// TIA Portal V16 export
// export: Created 2021-11-12T13:32:58.6971257Z, ExportSetting WithDefaults, DisplayName Totally Integrated Automation Portal, DisplayVersion V16 Update 3, DisplayName TIA Portal Version Control Interface, DisplayVersion V16 Update 2, DisplayName TIA Portal Openness, DisplayVersion V16 Update 3, DisplayName SINAMICS Startdrive Advanced, DisplayVersion V16 Update 5, DisplayName SINAMICS Startdrive G130, G150, S120, S150, SINAMICS MV, S210, DisplayVersion V16 Update 5, DisplayName SINAMICS Startdrive G110M, G120, G120C, G120D, G120P, G115D, DisplayVersion V16 Update 5, DisplayName STEP 7 Professional, DisplayVersion V16 Update 3, DisplayName STEP 7 Safety, DisplayVersion V16, DisplayName WinCC UA Professional, DisplayVersion V16 Update 3
FUNCTION_BLOCK "StationTHM1"   // FB80, LAD
{ S7_Optimized_Access := 'TRUE' }
VERSION : 0.1
// stored: AutoNumber true, IsIECCheckEnabled false, IsRetainMemResEnabled false, MemoryReserve 100, SetENOAutomatically false, UDAEnableTagReadback false
   VAR_INPUT
      IS_Inputs : "UDT_COMM_THM1_CRS";   // Input structure from blasting machine THM1
   END_VAR
   VAR_OUTPUT
      OS_Outputs : "UDT_COMM_CRS_THM1";   // Output structure for blasting machine THM1
      OS_Specific : "UDT_THM_Status_specific";   // Specific output structure for blasting machine THM1
   END_VAR
   VAR
      SF_Alarm1 : "STD_DI_Mon";
      SF_Alarm2 : "STD_DI_Mon";
      SF_Alarm3 : "STD_DI_Mon";
      SF_Alarm4 : "STD_DI_Mon";
      SF_Alarm5 : "STD_DI_Mon";
      SF_Alarm6 : "STD_DI_Mon";
      SF_Alarm7 : "STD_DI_Mon";
      SF_Alarm8 : "STD_DI_Mon";
      SS_Edge : Array[0..15] of Bool;   // Edge evalution
      SS_ParamTemp : Struct   // Structure of parameters
         PartType : Int;   // Conveyor speed setpoint
         ConvSpd : Int;   // THM1 - Transportation system speed setpoint
      END_STRUCT;
      SB1ParamChanged : Bool;   // Production paramaters changed trigger
   END_VAR
   VAR_TEMP
      TB1PwrOk : Bool;   // Station powered
      TB1SetParam : Bool;   // Set loaded parameters memory
   END_VAR
   VAR_TEMP   // added for the SCL form of the ladder/FBD networks
      _w1 : Bool;
      _w2 : Bool;
   END_VAR
BEGIN

REGION Network 1: *************** Alarms ***************
END_REGION

REGION Network 2: Power OK
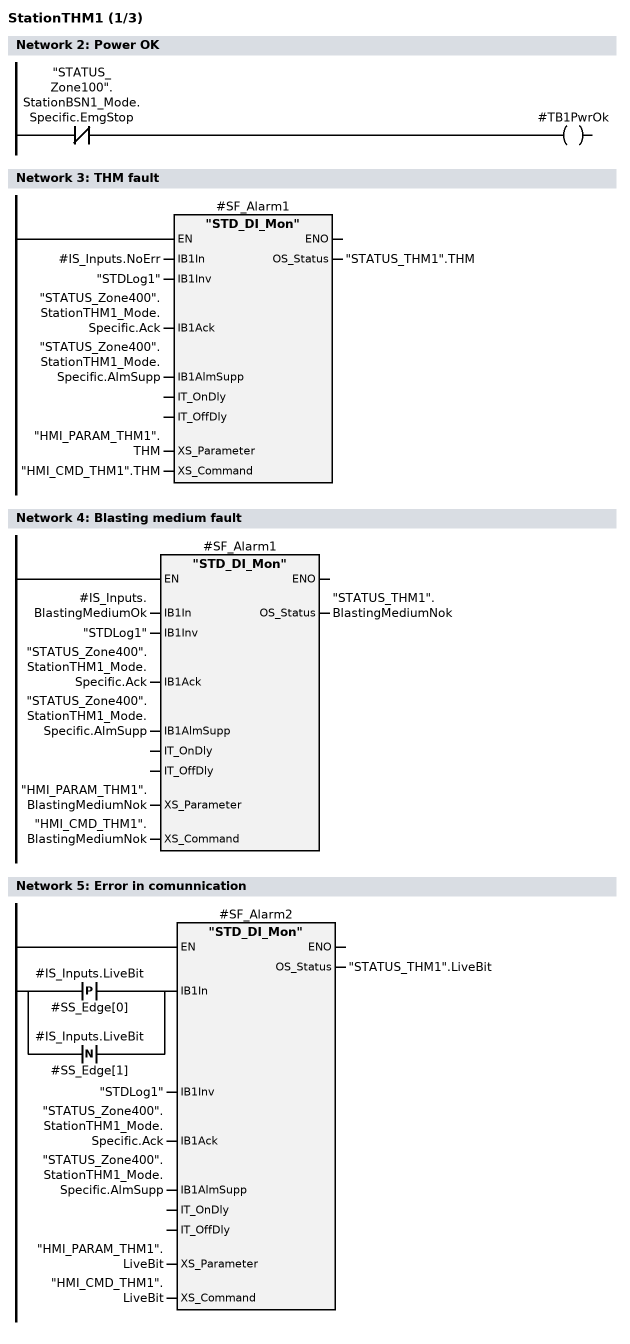
   RUNG wire#powerrail
      I_Contact( "STATUS_Zone100".StationBSN1_Mode.Specific.EmgStop )
      Coil( #TB1PwrOk )
   END_RUNG
   // the same network as SCL:
   #TB1PwrOk := NOT "STATUS_Zone100".StationBSN1_Mode.Specific.EmgStop;
END_REGION

REGION Network 3: THM fault
   RUNG wire#powerrail
      #SF_Alarm1(IB1In := #IS_Inputs.NoErr, IB1Inv := "STDLog1", IB1Ack := "STATUS_Zone400".StationTHM1_Mode.Specific.Ack, IB1AlmSupp := "STATUS_Zone400".StationTHM1_Mode.Specific.AlmSupp, IT_OnDly :=, IT_OffDly :=, XS_Parameter := "HMI_PARAM_THM1".THM, XS_Command := "HMI_CMD_THM1".THM, OS_Status => "STATUS_THM1".THM)
   END_RUNG
   // the same network as SCL:
   #SF_Alarm1(IB1In := #IS_Inputs.NoErr,   // "STD_DI_Mon"
              IB1Inv := "STDLog1",
              IB1Ack := "STATUS_Zone400".StationTHM1_Mode.Specific.Ack,
              IB1AlmSupp := "STATUS_Zone400".StationTHM1_Mode.Specific.AlmSupp,
              XS_Parameter := "HMI_PARAM_THM1".THM,
              XS_Command := "HMI_CMD_THM1".THM,
              OS_Status => "STATUS_THM1".THM);
END_REGION

REGION Network 4: Blasting medium fault
   RUNG wire#powerrail
      #SF_Alarm1(IB1In := #IS_Inputs.BlastingMediumOk, IB1Inv := "STDLog1", IB1Ack := "STATUS_Zone400".StationTHM1_Mode.Specific.Ack, IB1AlmSupp := "STATUS_Zone400".StationTHM1_Mode.Specific.AlmSupp, IT_OnDly :=, IT_OffDly :=, XS_Parameter := "HMI_PARAM_THM1".BlastingMediumNok, XS_Command := "HMI_CMD_THM1".BlastingMediumNok, OS_Status => "STATUS_THM1".BlastingMediumNok)
   END_RUNG
   // the same network as SCL:
   #SF_Alarm1(IB1In := #IS_Inputs.BlastingMediumOk,   // "STD_DI_Mon"
              IB1Inv := "STDLog1",
              IB1Ack := "STATUS_Zone400".StationTHM1_Mode.Specific.Ack,
              IB1AlmSupp := "STATUS_Zone400".StationTHM1_Mode.Specific.AlmSupp,
              XS_Parameter := "HMI_PARAM_THM1".BlastingMediumNok,
              XS_Command := "HMI_CMD_THM1".BlastingMediumNok,
              OS_Status => "STATUS_THM1".BlastingMediumNok);
END_REGION

REGION Network 5: Error in comunnication
   RUNG wire#powerrail
      #SF_Alarm2(IB1In := wire#w1, IB1Inv := "STDLog1", IB1Ack := "STATUS_Zone400".StationTHM1_Mode.Specific.Ack, IB1AlmSupp := "STATUS_Zone400".StationTHM1_Mode.Specific.AlmSupp, IT_OnDly :=, IT_OffDly :=, XS_Parameter := "HMI_PARAM_THM1".LiveBit, XS_Command := "HMI_CMD_THM1".LiveBit, OS_Status => "STATUS_THM1".LiveBit)
   END_RUNG
   RUNG wire#powerrail
      P_Contact(operand := #IS_Inputs.LiveBit, bit := #SS_Edge[0])
   END_RUNG wire#w1
   RUNG wire#powerrail
      N_Contact(operand := #IS_Inputs.LiveBit, bit := #SS_Edge[1])
   END_RUNG wire#w1
   // the same network as SCL:
   #_w1 := #IS_Inputs.LiveBit AND NOT #SS_Edge[0];   // rising edge of #IS_Inputs.LiveBit
   #SS_Edge[0] := #IS_Inputs.LiveBit;
   #_w2 := NOT #IS_Inputs.LiveBit AND #SS_Edge[1];   // falling edge of #IS_Inputs.LiveBit
   #SS_Edge[1] := #IS_Inputs.LiveBit;
   #SF_Alarm2(IB1In := #_w1 OR #_w2,   // "STD_DI_Mon"
              IB1Inv := "STDLog1",
              IB1Ack := "STATUS_Zone400".StationTHM1_Mode.Specific.Ack,
              IB1AlmSupp := "STATUS_Zone400".StationTHM1_Mode.Specific.AlmSupp,
              XS_Parameter := "HMI_PARAM_THM1".LiveBit,
              XS_Command := "HMI_CMD_THM1".LiveBit,
              OS_Status => "STATUS_THM1".LiveBit);
END_REGION

REGION Network 6: Production parameters not changed
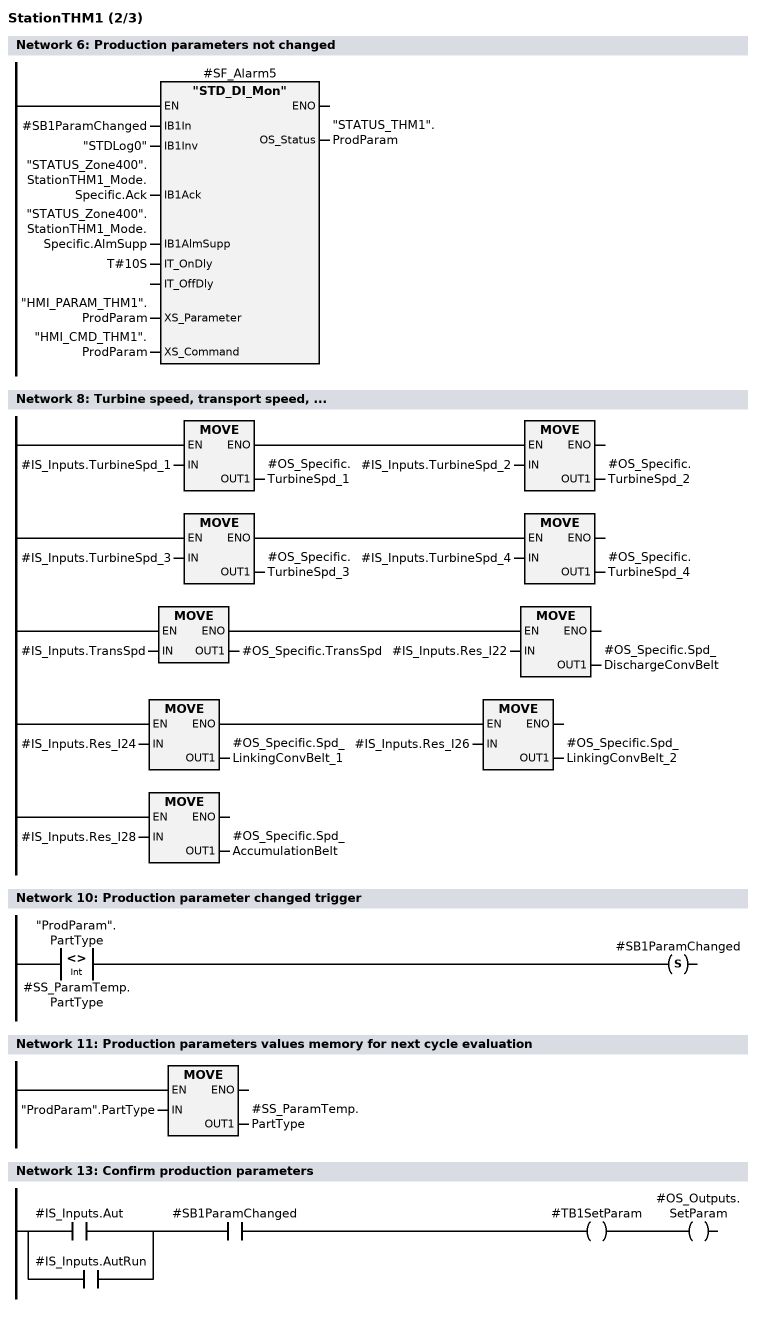
   RUNG wire#powerrail
      #SF_Alarm5(IB1In := #SB1ParamChanged, IB1Inv := "STDLog0", IB1Ack := "STATUS_Zone400".StationTHM1_Mode.Specific.Ack, IB1AlmSupp := "STATUS_Zone400".StationTHM1_Mode.Specific.AlmSupp, IT_OnDly := T#10S, IT_OffDly :=, XS_Parameter := "HMI_PARAM_THM1".ProdParam, XS_Command := "HMI_CMD_THM1".ProdParam, OS_Status => "STATUS_THM1".ProdParam)
   END_RUNG
   // the same network as SCL:
   #SF_Alarm5(IB1In := #SB1ParamChanged,   // "STD_DI_Mon"
              IB1Inv := "STDLog0",
              IB1Ack := "STATUS_Zone400".StationTHM1_Mode.Specific.Ack,
              IB1AlmSupp := "STATUS_Zone400".StationTHM1_Mode.Specific.AlmSupp,
              IT_OnDly := T#10S,
              XS_Parameter := "HMI_PARAM_THM1".ProdParam,
              XS_Command := "HMI_CMD_THM1".ProdParam,
              OS_Status => "STATUS_THM1".ProdParam);
END_REGION

REGION Network 7: *************** Statuses ***************
END_REGION

REGION Network 8: Turbine speed, transport speed, ...
   RUNG wire#powerrail
      Move(in := #IS_Inputs.TurbineSpd_1, out1 => #OS_Specific.TurbineSpd_1)
      Move(in := #IS_Inputs.TurbineSpd_2, out1 => #OS_Specific.TurbineSpd_2)
   END_RUNG
   RUNG wire#powerrail
      Move(in := #IS_Inputs.TurbineSpd_3, out1 => #OS_Specific.TurbineSpd_3)
      Move(in := #IS_Inputs.TurbineSpd_4, out1 => #OS_Specific.TurbineSpd_4)
   END_RUNG
   RUNG wire#powerrail
      Move(in := #IS_Inputs.TransSpd, out1 => #OS_Specific.TransSpd)
      Move(in := #IS_Inputs.Res_I22, out1 => #OS_Specific.Spd_DischargeConvBelt)
   END_RUNG
   RUNG wire#powerrail
      Move(in := #IS_Inputs.Res_I24, out1 => #OS_Specific.Spd_LinkingConvBelt_1)
      Move(in := #IS_Inputs.Res_I26, out1 => #OS_Specific.Spd_LinkingConvBelt_2)
   END_RUNG
   RUNG wire#powerrail
      Move(in := #IS_Inputs.Res_I28, out1 => #OS_Specific.Spd_AccumulationBelt)
   END_RUNG
   // the same network as SCL:
   #OS_Specific.TurbineSpd_1 := #IS_Inputs.TurbineSpd_1;
   #OS_Specific.TurbineSpd_2 := #IS_Inputs.TurbineSpd_2;
   #OS_Specific.TurbineSpd_3 := #IS_Inputs.TurbineSpd_3;
   #OS_Specific.TurbineSpd_4 := #IS_Inputs.TurbineSpd_4;
   #OS_Specific.TransSpd := #IS_Inputs.TransSpd;
   #OS_Specific.Spd_DischargeConvBelt := #IS_Inputs.Res_I22;
   #OS_Specific.Spd_LinkingConvBelt_1 := #IS_Inputs.Res_I24;
   #OS_Specific.Spd_LinkingConvBelt_2 := #IS_Inputs.Res_I26;
   #OS_Specific.Spd_AccumulationBelt := #IS_Inputs.Res_I28;
END_REGION

REGION Network 9: ************** Production parameters***************
END_REGION

REGION Network 10: Production parameter changed trigger
   RUNG wire#powerrail
      { S7_Templates := "SrcType := Int" } NE_Contact(in1 := "ProdParam".PartType, in2 := #SS_ParamTemp.PartType)
      S_Coil( #SB1ParamChanged )
   END_RUNG
   // the same network as SCL:
   IF "ProdParam".PartType <> #SS_ParamTemp.PartType THEN #SB1ParamChanged := TRUE; END_IF;
END_REGION

REGION Network 11: Production parameters values memory for next cycle evaluation
   RUNG wire#powerrail
      Move(in := "ProdParam".PartType, out1 => #SS_ParamTemp.PartType)
   END_RUNG
   // the same network as SCL:
   #SS_ParamTemp.PartType := "ProdParam".PartType;
END_REGION

REGION Network 12: Send production parameters to THM PLC
END_REGION

REGION Network 13: Confirm production parameters
   RUNG wire#powerrail
      Contact( #IS_Inputs.Aut )
      wire#w1
      Contact( #SB1ParamChanged )
      Coil( #TB1SetParam )
      Coil( #OS_Outputs.SetParam )
   END_RUNG
   RUNG wire#powerrail
      Contact( #IS_Inputs.AutRun )
   END_RUNG wire#w1
   // the same network as SCL:
   #TB1SetParam := (#IS_Inputs.Aut OR #IS_Inputs.AutRun) AND #SB1ParamChanged;
   #OS_Outputs.SetParam := #TB1SetParam;
END_REGION

REGION Network 14: Reset production parameter changed trigger
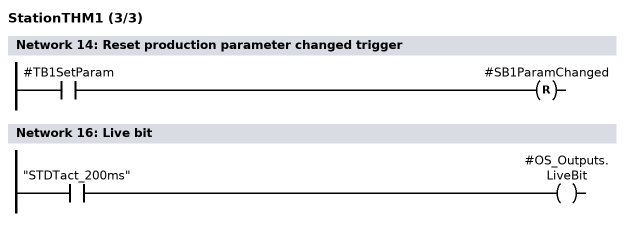
   RUNG wire#powerrail
      Contact( #TB1SetParam )
      R_Coil( #SB1ParamChanged )
   END_RUNG
   // the same network as SCL:
   IF #TB1SetParam THEN #SB1ParamChanged := FALSE; END_IF;
END_REGION

REGION Network 15: *************** Interface ***************
END_REGION

REGION Network 16: Live bit
   RUNG wire#powerrail
      Contact( "STDTact_200ms" )
      Coil( #OS_Outputs.LiveBit )
   END_RUNG
   // the same network as SCL:
   #OS_Outputs.LiveBit := "STDTact_200ms";
END_REGION
END_FUNCTION_BLOCK
